INTERFACE I_FIFO_Timestruct EXTENDS I_Universal_FIFO

METHOD MR_AddValue : BOOL
VAR_INPUT
		Value : TIMESTRUCT;
END_VAR
END_METHOD

PROPERTY oOldestValue : TIMESTRUCT
GET
END_GET
END_PROPERTY

END_INTERFACE

(* stored: Version 1.1.0.1, ProductVersion 3.1.4024.12
   Itf I_FIFO_Timestruct: Id {7bc79695-e5a3-41c2-a4f1-3687535dd940}
   Method MR_AddValue: Id {ee64d589-d615-454d-9d0f-cfb797aa7ee1}
   Property oOldestValue: Id {2b94cc3f-a587-4e8f-87f0-b190525260f2}
   Get Get: Id {344c5bc6-881f-442f-8846-84dd4f51410d} *)
